TYPE (* IEC61131-3, Table 14#5 *)
  (* Standard: 1131-3 *)
  (* Version 0.0, 6/4/2026, Schneider Electric, Template *)
  PACKAGE SE.Nereda;
  {SET_ATTRIBUTE(nxtDataType, uyyvlADWW18nMN04pyeUi3s8KgGwGCeiFv+F4pHVZt7rXg7S1fgYVV+sPWsFq9L1)}
  DeviceType : (
    Motor,
    Valve
  );
END_TYPE
